// TwinCAT 3 PLC project Lab_1
// ProgramVersion: 3.1.4022.4
// libraries:
//   Tc2_Standard, * (Beckhoff Automation GmbH)
//   Tc2_System, * (Beckhoff Automation GmbH)
//   Tc3_Module, * (Beckhoff Automation GmbH)
// project tree:
//   / GlobalTextList.TcGTLO, PlcTask.TcTTO, Visualization Manager.TcVMO (not stored)
//   POUs/ MAIN.TcPOU
//   VISUs/ Visualization.TcVIS
// real-time tasks:
//   TASK PlcTask: cycle T#10ms, priority 20, ADS port 350

CONFIGURATION Lab_1
    RESOURCE PLC ON TwinCAT3
        TASK PlcTask(INTERVAL := T#10ms, PRIORITY := 20);
        PROGRAM MAIN WITH PlcTask : MAIN;
    END_RESOURCE
END_CONFIGURATION

// ---- POUs/MAIN.TcPOU
PROGRAM MAIN
VAR
	//To attach variables to IO modules, it is needed to use "AT",
	// Inputs - I, Output - Q 
	bStart AT %I* 	: BOOL; 		// start button
	bLamp AT %Q*	: BOOL;			// Lamp 
	
	// Local variables without connecting to IO
	bStatus 		: BOOL;
	
END_VAR


// Switch on the lamp with push button in visualization.
bLamp := bStart;

END_PROGRAM

// ---- GlobalTextList.TcGTLO
TEXTLIST GlobalTextList
  102 = 'Start'
  277 = 'Start counting'
END_TEXTLIST

// ---- VISUs/Visualization.TcVIS
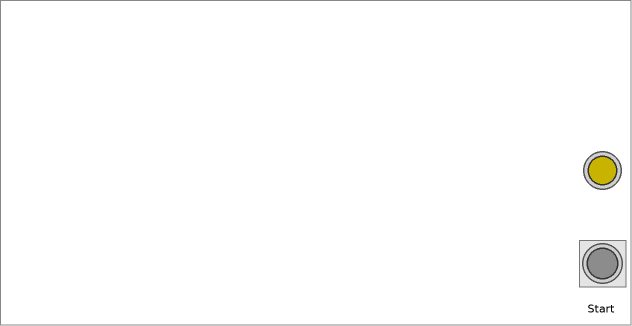
VISUALIZATION Visualization  // 632x326
    Lamp1 (580,148 45x45), variable: MAIN.bLamp, style: Lamp-Lamp1-Yellow
    PushSwitch (579,240 47x47), variable: MAIN.bStart, behaviour: TOGGLE, style: Switch-PushSwitch-Gray
    Label (572,294 58x30), "Start"
END_VISUALIZATION
